FUNCTION_BLOCK IORevPiCore (* Core module for Revolution Pi by KUNBUS GmbH *)
  (* Standard: 61499-2; Description: Copyright (c) 2018 fortiss GmbH This program and the accompanying materials are made available under the terms of the Eclipse Public License 2.0 which is available at https://www.eclipse.org/legal/epl-2.0/ SPDX-License-Identifier: EPL-2.0 *)
  (* Version 1.0, 2018-04-22, Jos?? Cabral, fortiss GmbH *)
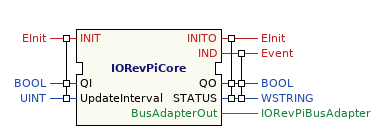
  EVENT_INPUT
    INIT : EInit WITH QI, UpdateInterval; (* Service Initialization *)
  END_EVENT
  EVENT_OUTPUT
    INITO : EInit WITH QO, STATUS; (* Initialization Confirm *)
    IND WITH QO, STATUS; (* Indication from Resource *)
  END_EVENT
  VAR_INPUT
    QI : BOOL; (* Event Input Qualifier *)
    UpdateInterval : UINT := 25; (* Update interval in Hz *)
  END_VAR
  VAR_OUTPUT
    QO : BOOL; (* Event Output Qualifier *)
    STATUS : WSTRING; (* Service Status *)
  END_VAR
  PLUGS
    BusAdapterOut : IORevPiBusAdapter;
  END_PLUGS
END_FUNCTION_BLOCK
